(* IEC 61131-3 sources: Word/plc-course/23-commissioning-and-troubleshooting/labs/solutions, 3 files *)

(* ---- 23-3-io-simulation.st ---- *)
(* Lab 23-3: I/O simulation layer for checkout - transfer pump P-101.
   Module 23 (Commissioning and troubleshooting). REFERENCE SOLUTION - try the lab yourself first.

   Every field input passes through a small simulation block before the
   application logic sees it. During a FAT or I/O checkout a tester can put a
   point into simulation from the HMI and type a value, but only while the
   "simulation permitted" key switch is on. A lamp and a counter show that
   simulation is active. Training exercise only: a real plant needs site rules
   for who may simulate what, and simulation must never bypass a safety function. *)

TYPE
  ST_SimDI : STRUCT
    Enable : BOOL;  (* HMI: put this point into simulation *)
    Value  : BOOL;  (* HMI: simulated value *)
  END_STRUCT;
  ST_SimAI : STRUCT
    Enable : BOOL;  (* HMI: put this point into simulation *)
    Value  : REAL;  (* HMI: simulated value in engineering units *)
  END_STRUCT;
END_TYPE

(* One digital input point. Call it every scan, before the logic that uses Value. *)
FUNCTION_BLOCK FB_SimDI
  VAR_INPUT
    Live   : BOOL;  (* value from the field *)
    Permit : BOOL;  (* simulation permitted (key switch) *)
  END_VAR
  VAR_IN_OUT
    Sim : ST_SimDI;  (* this point's HMI simulation tags *)
  END_VAR
  VAR_OUTPUT
    Value  : BOOL;  (* value for the application logic *)
    Active : BOOL;  (* this point is being simulated *)
  END_VAR
  VAR
    WasActive : BOOL;
  END_VAR

  IF NOT Permit THEN
    Sim.Enable := FALSE;       (* no key: refuse and clear any request *)
  END_IF;
  Active := Sim.Enable;
  IF Active AND NOT WasActive THEN
    Sim.Value := Live;         (* bumpless start: begin from the live value *)
  END_IF;
  WasActive := Active;
  IF Active THEN
    Value := Sim.Value;
  ELSE
    Value := Live;
  END_IF;
END_FUNCTION_BLOCK

(* One analog input point, in engineering units. Same rules as FB_SimDI. *)
FUNCTION_BLOCK FB_SimAI
  VAR_INPUT
    Live   : REAL;
    Permit : BOOL;
  END_VAR
  VAR_IN_OUT
    Sim : ST_SimAI;
  END_VAR
  VAR_OUTPUT
    Value  : REAL;
    Active : BOOL;
  END_VAR
  VAR
    WasActive : BOOL;
  END_VAR

  IF NOT Permit THEN
    Sim.Enable := FALSE;
  END_IF;
  Active := Sim.Enable;
  IF Active AND NOT WasActive THEN
    Sim.Value := Live;
  END_IF;
  WasActive := Active;
  IF Active THEN
    Value := Sim.Value;
  ELSE
    Value := Live;
  END_IF;
END_FUNCTION_BLOCK

PROGRAM PumpCheckout
  VAR (* I/O - addresses follow the OpenPLC convention *)
    LSL101_NC AT %IX0.0 : BOOL;  (* LSL-101 low-level switch, NC: TRUE while level is above it *)
    P101RunFB AT %IX0.1 : BOOL;  (* P-101 contactor auxiliary contact: TRUE = running *)
    SimKeySW  AT %IX0.2 : BOOL;  (* key switch "simulation permitted" (commissioning only) *)
    ResetPB   AT %IX0.3 : BOOL;  (* fault reset push-button, NO *)
    LT101Raw  AT %IW0   : INT;   (* LT-101 tank level, 4-20 mA input: 0..27648 = 0..100 % *)
    P101Run   AT %QX0.0 : BOOL;  (* P-101 contactor coil *)
    SimLamp   AT %QX0.1 : BOOL;  (* amber lamp: simulation active *)
    P101Fault AT %QX0.2 : BOOL;  (* red lamp: P-101 failed to start *)
  END_VAR
  VAR (* HMI simulation tags, one structure per point *)
    SimLSL101 : ST_SimDI;
    SimP101FB : ST_SimDI;
    SimLT101  : ST_SimAI;
  END_VAR
  VAR (* processed values: the ONLY input values the application logic uses *)
    LSL101_OK   : BOOL;
    P101Running : BOOL;
    LT101_Pct   : REAL;
  END_VAR
  VAR (* simulation status for the HMI banner *)
    SimActive : BOOL;
    SimCount  : INT;
  END_VAR
  VAR (* internal *)
    LT101_Live : REAL;
    SimLSL     : FB_SimDI;
    SimFB      : FB_SimDI;
    SimLT      : FB_SimAI;
    PumpDemand : BOOL;
    FbTimer    : TON;
  END_VAR

  (* ==== SIMULATION LAYER: runs first, so the logic sees this scan's values ==== *)
  LT101_Live := INT_TO_REAL(LT101Raw) * 100.0 / 27648.0;

  SimLSL(Live := LSL101_NC, Permit := SimKeySW, Sim := SimLSL101);
  SimFB(Live := P101RunFB, Permit := SimKeySW, Sim := SimP101FB);
  SimLT(Live := LT101_Live, Permit := SimKeySW, Sim := SimLT101);

  LSL101_OK := SimLSL.Value;
  P101Running := SimFB.Value;
  LT101_Pct := SimLT.Value;

  SimCount := 0;
  IF SimLSL.Active THEN SimCount := SimCount + 1; END_IF;
  IF SimFB.Active THEN SimCount := SimCount + 1; END_IF;
  IF SimLT.Active THEN SimCount := SimCount + 1; END_IF;
  SimActive := SimCount > 0;
  SimLamp := SimActive;

  (* ==== APPLICATION LOGIC (given; uses processed values only) ==== *)
  (* Level control with hysteresis: start at 60 %, stop at 20 % *)
  IF LT101_Pct >= 60.0 THEN
    PumpDemand := TRUE;
  ELSIF LT101_Pct <= 20.0 THEN
    PumpDemand := FALSE;
  END_IF;

  (* Start failure: commanded but no running feedback within 2 s *)
  FbTimer(IN := P101Run AND NOT P101Running, PT := T#2s);
  IF FbTimer.Q THEN
    P101Fault := TRUE;
  ELSIF ResetPB THEN
    P101Fault := FALSE;
  END_IF;

  (* Command: demand AND dry-run protection AND no fault *)
  P101Run := PumpDemand AND LSL101_OK AND NOT P101Fault;
END_PROGRAM

CONFIGURATION Config0
  RESOURCE Res0 ON PLC
    TASK MainTask(INTERVAL := T#10ms, PRIORITY := 0);
    PROGRAM Inst0 WITH MainTask : PumpCheckout;
  END_RESOURCE
END_CONFIGURATION

(* ---- 23-1-find-the-bugs.st ---- *)
(* Lab 23-1: Find the bugs - transfer conveyor with jog and jam detection.
   Module 23 (Commissioning and troubleshooting). REFERENCE SOLUTION - try the lab yourself first.

   This is the starter program with its three bugs fixed. Each fix is marked
   "FIX 1", "FIX 2" or "FIX 3" so you can compare it with your own repair.
   Everything else is unchanged: in a real plant you fix the fault, not rewrite
   the program. *)

PROGRAM TransferConveyor
  VAR (* I/O - addresses follow the OpenPLC convention *)
    StartPB       AT %IX0.0 : BOOL;  (* Start push-button, NO: TRUE while pressed *)
    StopPB_NC     AT %IX0.1 : BOOL;  (* Stop push-button, NC: TRUE while NOT pressed *)
    JogPB         AT %IX0.2 : BOOL;  (* Jog push-button, NO: conveyor runs only while held *)
    JamPE         AT %IX0.3 : BOOL;  (* Jam photo-eye at the discharge: TRUE while the beam is blocked *)
    ResetPB       AT %IX0.4 : BOOL;  (* Fault reset push-button, NO *)
    OverloadOK_NC AT %IX0.5 : BOOL;  (* Motor overload relay auxiliary contact, NC: TRUE while healthy *)
    ConveyorMotor AT %QX0.0 : BOOL;  (* Conveyor motor contactor coil *)
    RunLamp       AT %QX0.1 : BOOL;  (* Green lamp: running in automatic *)
    FaultLamp     AT %QX0.2 : BOOL;  (* Red lamp: a fault is latched *)
  END_VAR
  VAR (* internal *)
    RunLatch : BOOL;  (* automatic run, sealed in by Start *)
    JogRun   : BOOL;  (* jog command *)
    Fault    : BOOL;  (* latched fault: jam or motor overload *)
    JamTimer : TON;   (* photo-eye blocked for too long while running = jam *)
  END_VAR

  (* ---- 1. Jam detection -------------------------------------------------
     FIX 2: the timer is called on EVERY scan, outside any IF. The running
     condition has moved into IN, so the timer resets as soon as the conveyor
     stops or the beam clears. A timer that is not called cannot reset: in the
     starter it kept its old state while the conveyor was stopped. *)
  JamTimer(IN := RunLatch AND JamPE, PT := T#3s);

  (* ---- 2. Fault latch: set by the cause, reset only when the cause has gone *)
  IF JamTimer.Q OR NOT OverloadOK_NC THEN
    Fault := TRUE;
  ELSIF ResetPB AND NOT JamPE AND OverloadOK_NC THEN
    Fault := FALSE;
  END_IF;

  (* ---- 3. Automatic run latch --------------------------------------------
     FIX 3: a fault now drops the run latch. In the starter the latch stayed
     set during a fault, so pressing Reset restarted the conveyor by itself. *)
  RunLatch := (StartPB OR RunLatch) AND StopPB_NC AND NOT Fault;

  (* ---- 4. Jog for maintenance: momentary, only when stopped and healthy *)
  JogRun := JogPB AND StopPB_NC AND NOT RunLatch AND NOT Fault;

  (* ---- 5. Outputs --------------------------------------------------------
     FIX 1: the motor output is written in exactly ONE place. In the starter it
     was assigned twice ("double coil") and the jog line, being last, won. *)
  ConveyorMotor := RunLatch OR JogRun;
  RunLamp := RunLatch;
  FaultLamp := Fault;
END_PROGRAM

CONFIGURATION Config0
  RESOURCE Res0 ON PLC
    TASK MainTask(INTERVAL := T#10ms, PRIORITY := 0);
    PROGRAM Inst0 WITH MainTask : TransferConveyor;
  END_RESOURCE
END_CONFIGURATION

(* ---- 23-2-subtle-faults.st ---- *)
(* Lab 23-2: Subtle faults - drum filling station.
   Module 23 (Commissioning and troubleshooting). REFERENCE SOLUTION - try the lab yourself first.

   The starter's three faults are fixed here and marked "FIX 1", "FIX 2", "FIX 3".
   None of them shows up in a quick bench test: one needs the HMI, one needs a
   busy shift and one needs a power cut in the middle of a fill. *)

TYPE
  E_FillStep : (Idle, Filling, Done);
END_TYPE

PROGRAM DrumFiller
  VAR (* I/O - addresses follow the OpenPLC convention *)
    StartPB       AT %IX0.0 : BOOL;  (* Start push-button, NO *)
    StopPB_NC     AT %IX0.1 : BOOL;  (* Stop push-button, NC: TRUE while NOT pressed *)
    DrumPresentPX AT %IX0.2 : BOOL;  (* Proximity switch: a drum is in position on the scale *)
    WeightRaw     AT %IW0   : INT;   (* Scale transmitter via 4-20 mA input: 0..27648 = 0..300 kg *)
    FillValve     AT %QX0.0 : BOOL;  (* Fill valve solenoid, spring-return: de-energised = closed *)
    DoneLamp      AT %QX0.1 : BOOL;  (* White lamp: drum full, remove it *)
  END_VAR
  VAR (* HMI commands: the HMI writes TRUE, the PLC clears them (momentary) *)
    HmiStartCmd      : BOOL;  (* HMI "Start fill" button *)
    HmiResetCountCmd : BOOL;  (* HMI "Reset shift count" button *)
  END_VAR
  VAR (* HMI display values *)
    Weight_kg : REAL;  (* gross weight on the scale *)
    TotalKg   : DINT;  (* nominal kg filled this shift = DrumCount x 200 kg *)
  END_VAR
  VAR RETAIN (* must survive a power cut *)
    DrumCount : INT;   (* drums filled this shift *)
  END_VAR
  VAR (* internal *)
    (* FIX 3 (part 1): the step is no longer declared RETAIN. There is no
       reason to remember it through a power cut. But see the start-up section:
       some platforms keep every value anyway, so the code must not rely on it. *)
    FillStep    : E_FillStep := Idle;
    StartupDone : BOOL;  (* non-retentive: FALSE again after every PLC start *)
    StartReq    : BOOL;
    Tare_kg     : REAL;  (* weight of the empty drum, captured at the start *)
    Net_kg      : REAL;  (* product added so far *)
  END_VAR
  VAR CONSTANT
    TargetNet_kg   : REAL := 200.0;  (* product per drum *)
    EmptyMax_kg    : REAL := 50.0;   (* heavier than this = not an empty drum *)
    DrumNominal_kg : INT := 200;     (* used for the shift total *)
  END_VAR

  (* ---- 0. Start-up ----------------------------------------------------------
     FIX 3 (part 2): on the first scan after every PLC start the sequence is
     forced to Idle, whatever the memory holds, BEFORE any logic that drives an
     output. A fill interrupted by a power cut is never resumed automatically:
     the tare was lost and nobody has checked the drum. The retained shift count
     is deliberately left alone. *)
  IF NOT StartupDone THEN
    FillStep := Idle;
    StartupDone := TRUE;
  END_IF;

  (* ---- 1. Scale: raw counts to kilograms (Module 14) *)
  Weight_kg := INT_TO_REAL(WeightRaw) * 300.0 / 27648.0;

  (* ---- 2. Start request from the panel push-button or the HMI *)
  StartReq := StartPB OR HmiStartCmd;

  (* ---- 3. Fill sequence *)
  CASE FillStep OF
    Idle:
      (* Start only with a healthy stop circuit and an EMPTY drum in place *)
      IF StartReq AND StopPB_NC AND DrumPresentPX AND (Weight_kg < EmptyMax_kg) THEN
        Tare_kg := Weight_kg;
        Net_kg := 0.0;
        FillStep := Filling;
      END_IF;

    Filling:
      Net_kg := Weight_kg - Tare_kg;
      IF NOT StopPB_NC OR NOT DrumPresentPX THEN
        FillStep := Idle;                      (* abort: this drum is not counted *)
      ELSIF Net_kg >= TargetNet_kg THEN
        DrumCount := DrumCount + 1;
        FillStep := Done;
      END_IF;

    Done:
      IF NOT DrumPresentPX THEN            (* full drum taken away *)
        FillStep := Idle;
      END_IF;
  END_CASE;

  (* ---- 4. Shift totals *)
  IF HmiResetCountCmd THEN
    DrumCount := 0;
  END_IF;
  (* FIX 2: convert to DINT FIRST, then multiply. In the starter the product
     DrumCount * 200 was an INT and overflowed at 164 drums (32 800 kg), before
     INT_TO_DINT ever saw it. *)
  TotalKg := INT_TO_DINT(DrumCount) * INT_TO_DINT(DrumNominal_kg);

  (* ---- 5. Momentary HMI commands are cleared by the PLC.
     FIX 1: this happens AFTER the logic that reads them. On OpenPLC (and in
     plctest) the HMI writes between scans, so clearing them at the top of the
     program (as the starter did) wiped every command before the logic could
     see it. Clearing them every scan, accepted or not, means a refused command
     is never remembered. On a controller whose communications can write a tag
     part-way through a scan, the more robust pattern is to copy each command
     into an internal bit and clear it in the next statement, at the top, and
     then use only the copy. *)
  HmiStartCmd := FALSE;
  HmiResetCountCmd := FALSE;

  (* ---- 6. Outputs, written once, from the step *)
  FillValve := (FillStep = Filling);
  DoneLamp := (FillStep = Done);
END_PROGRAM

CONFIGURATION Config0
  RESOURCE Res0 ON PLC
    TASK MainTask(INTERVAL := T#10ms, PRIORITY := 0);
    PROGRAM Inst0 WITH MainTask : DrumFiller;
  END_RESOURCE
END_CONFIGURATION
